D13998	WORD	Память для хранения названий рецептов. Задание 160. Символ 24
D13999	WORD	Память для хранения названий рецептов. Задание 160. Символ 25
D14000	WORD	Память для хранения названий рецептов. Задание 161. Символ 1
D14001	WORD	Память для хранения названий рецептов. Задание 161. Символ 2
D14002	WORD	Память для хранения названий рецептов. Задание 161. Символ 3
D14003	WORD	Память для хранения названий рецептов. Задание 161. Символ 4
D14004	WORD	Память для хранения названий рецептов. Задание 161. Символ 5
D14005	WORD	Память для хранения названий рецептов. Задание 161. Символ 6
D14006	WORD	Память для хранения названий рецептов. Задание 161. Символ 7
D14007	WORD	Память для хранения названий рецептов. Задание 161. Символ 8
D14008	WORD	Память для хранения названий рецептов. Задание 161. Символ 9
D14009	WORD	Память для хранения названий рецептов. Задание 161. Символ 10
D14010	WORD	Память для хранения названий рецептов. Задание 161. Символ 11
D14011	WORD	Память для хранения названий рецептов. Задание 161. Символ 12
D14012	WORD	Память для хранения названий рецептов. Задание 161. Символ 13
D14013	WORD	Память для хранения названий рецептов. Задание 161. Символ 14
D14014	WORD	Память для хранения названий рецептов. Задание 161. Символ 15
D14015	WORD	Память для хранения названий рецептов. Задание 161. Символ 16
D14016	WORD	Память для хранения названий рецептов. Задание 161. Символ 17
D14017	WORD	Память для хранения названий рецептов. Задание 161. Символ 18
D14018	WORD	Память для хранения названий рецептов. Задание 161. Символ 19
D14019	WORD	Память для хранения названий рецептов. Задание 161. Символ 20
D14020	WORD	Память для хранения названий рецептов. Задание 161. Символ 21
D14021	WORD	Память для хранения названий рецептов. Задание 161. Символ 22
D14022	WORD	Память для хранения названий рецептов. Задание 161. Символ 23
D14023	WORD	Память для хранения названий рецептов. Задание 161. Символ 24
D14024	WORD	Память для хранения названий рецептов. Задание 161. Символ 25
D14025	WORD	Память для хранения названий рецептов. Задание 162. Символ 1
D14026	WORD	Память для хранения названий рецептов. Задание 162. Символ 2
D14027	WORD	Память для хранения названий рецептов. Задание 162. Символ 3
D14028	WORD	Память для хранения названий рецептов. Задание 162. Символ 4
D14029	WORD	Память для хранения названий рецептов. Задание 162. Символ 5
D14030	WORD	Память для хранения названий рецептов. Задание 162. Символ 6
D14031	WORD	Память для хранения названий рецептов. Задание 162. Символ 7
D14032	WORD	Память для хранения названий рецептов. Задание 162. Символ 8
D14033	WORD	Память для хранения названий рецептов. Задание 162. Символ 9
D14034	WORD	Память для хранения названий рецептов. Задание 162. Символ 10
D14035	WORD	Память для хранения названий рецептов. Задание 162. Символ 11
D14036	WORD	Память для хранения названий рецептов. Задание 162. Символ 12
D14037	WORD	Память для хранения названий рецептов. Задание 162. Символ 13
D14038	WORD	Память для хранения названий рецептов. Задание 162. Символ 14
D14039	WORD	Память для хранения названий рецептов. Задание 162. Символ 15
D14040	WORD	Память для хранения названий рецептов. Задание 162. Символ 16
D14041	WORD	Память для хранения названий рецептов. Задание 162. Символ 17
D14042	WORD	Память для хранения названий рецептов. Задание 162. Символ 18
D14043	WORD	Память для хранения названий рецептов. Задание 162. Символ 19
D14044	WORD	Память для хранения названий рецептов. Задание 162. Символ 20
D14045	WORD	Память для хранения названий рецептов. Задание 162. Символ 21
D14046	WORD	Память для хранения названий рецептов. Задание 162. Символ 22
D14047	WORD	Память для хранения названий рецептов. Задание 162. Символ 23
D14048	WORD	Память для хранения названий рецептов. Задание 162. Символ 24
D14049	WORD	Память для хранения названий рецептов. Задание 162. Символ 25
D14050	WORD	Память для хранения названий рецептов. Задание 163. Символ 1
D14051	WORD	Память для хранения названий рецептов. Задание 163. Символ 2
D14052	WORD	Память для хранения названий рецептов. Задание 163. Символ 3
D14053	WORD	Память для хранения названий рецептов. Задание 163. Символ 4
D14054	WORD	Память для хранения названий рецептов. Задание 163. Символ 5
D14055	WORD	Память для хранения названий рецептов. Задание 163. Символ 6
D14056	WORD	Память для хранения названий рецептов. Задание 163. Символ 7
D14057	WORD	Память для хранения названий рецептов. Задание 163. Символ 8
D14058	WORD	Память для хранения названий рецептов. Задание 163. Символ 9
D14059	WORD	Память для хранения названий рецептов. Задание 163. Символ 10
D14060	WORD	Память для хранения названий рецептов. Задание 163. Символ 11
D14061	WORD	Память для хранения названий рецептов. Задание 163. Символ 12
D14062	WORD	Память для хранения названий рецептов. Задание 163. Символ 13
D14063	WORD	Память для хранения названий рецептов. Задание 163. Символ 14
D14064	WORD	Память для хранения названий рецептов. Задание 163. Символ 15
D14065	WORD	Память для хранения названий рецептов. Задание 163. Символ 16
D14066	WORD	Память для хранения названий рецептов. Задание 163. Символ 17
D14067	WORD	Память для хранения названий рецептов. Задание 163. Символ 18
D14068	WORD	Память для хранения названий рецептов. Задание 163. Символ 19
D14069	WORD	Память для хранения названий рецептов. Задание 163. Символ 20
D14070	WORD	Память для хранения названий рецептов. Задание 163. Символ 21
D14071	WORD	Память для хранения названий рецептов. Задание 163. Символ 22
D14072	WORD	Память для хранения названий рецептов. Задание 163. Символ 23
D14073	WORD	Память для хранения названий рецептов. Задание 163. Символ 24
D14074	WORD	Память для хранения названий рецептов. Задание 163. Символ 25
D14075	WORD	Память для хранения названий рецептов. Задание 164. Символ 1
D14076	WORD	Память для хранения названий рецептов. Задание 164. Символ 2
D14077	WORD	Память для хранения названий рецептов. Задание 164. Символ 3
D14078	WORD	Память для хранения названий рецептов. Задание 164. Символ 4
D14079	WORD	Память для хранения названий рецептов. Задание 164. Символ 5
D14080	WORD	Память для хранения названий рецептов. Задание 164. Символ 6
D14081	WORD	Память для хранения названий рецептов. Задание 164. Символ 7
D14082	WORD	Память для хранения названий рецептов. Задание 164. Символ 8
D14083	WORD	Память для хранения названий рецептов. Задание 164. Символ 9
D14084	WORD	Память для хранения названий рецептов. Задание 164. Символ 10
D14085	WORD	Память для хранения названий рецептов. Задание 164. Символ 11
D14086	WORD	Память для хранения названий рецептов. Задание 164. Символ 12
D14087	WORD	Память для хранения названий рецептов. Задание 164. Символ 13
D14088	WORD	Память для хранения названий рецептов. Задание 164. Символ 14
D14089	WORD	Память для хранения названий рецептов. Задание 164. Символ 15
D14090	WORD	Память для хранения названий рецептов. Задание 164. Символ 16
D14091	WORD	Память для хранения названий рецептов. Задание 164. Символ 17
D14092	WORD	Память для хранения названий рецептов. Задание 164. Символ 18
D14093	WORD	Память для хранения названий рецептов. Задание 164. Символ 19
D14094	WORD	Память для хранения названий рецептов. Задание 164. Символ 20
D14095	WORD	Память для хранения названий рецептов. Задание 164. Символ 21
D14096	WORD	Память для хранения названий рецептов. Задание 164. Символ 22
D14097	WORD	Память для хранения названий рецептов. Задание 164. Символ 23
D14098	WORD	Память для хранения названий рецептов. Задание 164. Символ 24
D14099	WORD	Память для хранения названий рецептов. Задание 164. Символ 25
D14100	WORD	Память для хранения названий рецептов. Задание 165. Символ 1
D14101	WORD	Память для хранения названий рецептов. Задание 165. Символ 2
D14102	WORD	Память для хранения названий рецептов. Задание 165. Символ 3
D14103	WORD	Память для хранения названий рецептов. Задание 165. Символ 4
D14104	WORD	Память для хранения названий рецептов. Задание 165. Символ 5
D14105	WORD	Память для хранения названий рецептов. Задание 165. Символ 6
D14106	WORD	Память для хранения названий рецептов. Задание 165. Символ 7
D14107	WORD	Память для хранения названий рецептов. Задание 165. Символ 8
D14108	WORD	Память для хранения названий рецептов. Задание 165. Символ 9
D14109	WORD	Память для хранения названий рецептов. Задание 165. Символ 10
D14110	WORD	Память для хранения названий рецептов. Задание 165. Символ 11
D14111	WORD	Память для хранения названий рецептов. Задание 165. Символ 12
D14112	WORD	Память для хранения названий рецептов. Задание 165. Символ 13
D14113	WORD	Память для хранения названий рецептов. Задание 165. Символ 14
D14114	WORD	Память для хранения названий рецептов. Задание 165. Символ 15
D14115	WORD	Память для хранения названий рецептов. Задание 165. Символ 16
D14116	WORD	Память для хранения названий рецептов. Задание 165. Символ 17
D14117	WORD	Память для хранения названий рецептов. Задание 165. Символ 18
D14118	WORD	Память для хранения названий рецептов. Задание 165. Символ 19
D14119	WORD	Память для хранения названий рецептов. Задание 165. Символ 20
D14120	WORD	Память для хранения названий рецептов. Задание 165. Символ 21
D14121	WORD	Память для хранения названий рецептов. Задание 165. Символ 22
D14122	WORD	Память для хранения названий рецептов. Задание 165. Символ 23
D14123	WORD	Память для хранения названий рецептов. Задание 165. Символ 24
D14124	WORD	Память для хранения названий рецептов. Задание 165. Символ 25
D14125	WORD	Память для хранения названий рецептов. Задание 166. Символ 1
D14126	WORD	Память для хранения названий рецептов. Задание 166. Символ 2
D14127	WORD	Память для хранения названий рецептов. Задание 166. Символ 3
D14128	WORD	Память для хранения названий рецептов. Задание 166. Символ 4
D14129	WORD	Память для хранения названий рецептов. Задание 166. Символ 5
D14130	WORD	Память для хранения названий рецептов. Задание 166. Символ 6
D14131	WORD	Память для хранения названий рецептов. Задание 166. Символ 7
D14132	WORD	Память для хранения названий рецептов. Задание 166. Символ 8
D14133	WORD	Память для хранения названий рецептов. Задание 166. Символ 9
D14134	WORD	Память для хранения названий рецептов. Задание 166. Символ 10
D14135	WORD	Память для хранения названий рецептов. Задание 166. Символ 11
D14136	WORD	Память для хранения названий рецептов. Задание 166. Символ 12
D14137	WORD	Память для хранения названий рецептов. Задание 166. Символ 13
D14138	WORD	Память для хранения названий рецептов. Задание 166. Символ 14
D14139	WORD	Память для хранения названий рецептов. Задание 166. Символ 15
D14140	WORD	Память для хранения названий рецептов. Задание 166. Символ 16
D14141	WORD	Память для хранения названий рецептов. Задание 166. Символ 17
D14142	WORD	Память для хранения названий рецептов. Задание 166. Символ 18
D14143	WORD	Память для хранения названий рецептов. Задание 166. Символ 19
D14144	WORD	Память для хранения названий рецептов. Задание 166. Символ 20
D14145	WORD	Память для хранения названий рецептов. Задание 166. Символ 21
D14146	WORD	Память для хранения названий рецептов. Задание 166. Символ 22
D14147	WORD	Память для хранения названий рецептов. Задание 166. Символ 23
D14148	WORD	Память для хранения названий рецептов. Задание 166. Символ 24
D14149	WORD	Память для хранения названий рецептов. Задание 166. Символ 25
D14150	WORD	Память для хранения названий рецептов. Задание 167. Символ 1
D14151	WORD	Память для хранения названий рецептов. Задание 167. Символ 2
D14152	WORD	Память для хранения названий рецептов. Задание 167. Символ 3
D14153	WORD	Память для хранения названий рецептов. Задание 167. Символ 4
D14154	WORD	Память для хранения названий рецептов. Задание 167. Символ 5
D14155	WORD	Память для хранения названий рецептов. Задание 167. Символ 6
D14156	WORD	Память для хранения названий рецептов. Задание 167. Символ 7
D14157	WORD	Память для хранения названий рецептов. Задание 167. Символ 8
D14158	WORD	Память для хранения названий рецептов. Задание 167. Символ 9
D14159	WORD	Память для хранения названий рецептов. Задание 167. Символ 10
D14160	WORD	Память для хранения названий рецептов. Задание 167. Символ 11
D14161	WORD	Память для хранения названий рецептов. Задание 167. Символ 12
D14162	WORD	Память для хранения названий рецептов. Задание 167. Символ 13
D14163	WORD	Память для хранения названий рецептов. Задание 167. Символ 14
D14164	WORD	Память для хранения названий рецептов. Задание 167. Символ 15
D14165	WORD	Память для хранения названий рецептов. Задание 167. Символ 16
D14166	WORD	Память для хранения названий рецептов. Задание 167. Символ 17
D14167	WORD	Память для хранения названий рецептов. Задание 167. Символ 18
D14168	WORD	Память для хранения названий рецептов. Задание 167. Символ 19
D14169	WORD	Память для хранения названий рецептов. Задание 167. Символ 20
D14170	WORD	Память для хранения названий рецептов. Задание 167. Символ 21
D14171	WORD	Память для хранения названий рецептов. Задание 167. Символ 22
D14172	WORD	Память для хранения названий рецептов. Задание 167. Символ 23
D14173	WORD	Память для хранения названий рецептов. Задание 167. Символ 24
D14174	WORD	Память для хранения названий рецептов. Задание 167. Символ 25
D14175	WORD	Память для хранения названий рецептов. Задание 168. Символ 1
D14176	WORD	Память для хранения названий рецептов. Задание 168. Символ 2
D14177	WORD	Память для хранения названий рецептов. Задание 168. Символ 3
D14178	WORD	Память для хранения названий рецептов. Задание 168. Символ 4
D14179	WORD	Память для хранения названий рецептов. Задание 168. Символ 5
D14180	WORD	Память для хранения названий рецептов. Задание 168. Символ 6
D14181	WORD	Память для хранения названий рецептов. Задание 168. Символ 7
D14182	WORD	Память для хранения названий рецептов. Задание 168. Символ 8
D14183	WORD	Память для хранения названий рецептов. Задание 168. Символ 9
D14184	WORD	Память для хранения названий рецептов. Задание 168. Символ 10
D14185	WORD	Память для хранения названий рецептов. Задание 168. Символ 11
D14186	WORD	Память для хранения названий рецептов. Задание 168. Символ 12
D14187	WORD	Память для хранения названий рецептов. Задание 168. Символ 13
D14188	WORD	Память для хранения названий рецептов. Задание 168. Символ 14
D14189	WORD	Память для хранения названий рецептов. Задание 168. Символ 15
D14190	WORD	Память для хранения названий рецептов. Задание 168. Символ 16
D14191	WORD	Память для хранения названий рецептов. Задание 168. Символ 17
D14192	WORD	Память для хранения названий рецептов. Задание 168. Символ 18
D14193	WORD	Память для хранения названий рецептов. Задание 168. Символ 19
D14194	WORD	Память для хранения названий рецептов. Задание 168. Символ 20
D14195	WORD	Память для хранения названий рецептов. Задание 168. Символ 21
D14196	WORD	Память для хранения названий рецептов. Задание 168. Символ 22
D14197	WORD	Память для хранения названий рецептов. Задание 168. Символ 23
D14198	WORD	Память для хранения названий рецептов. Задание 168. Символ 24
D14199	WORD	Память для хранения названий рецептов. Задание 168. Символ 25
D14200	WORD	Память для хранения названий рецептов. Задание 169. Символ 1
D14201	WORD	Память для хранения названий рецептов. Задание 169. Символ 2
D14202	WORD	Память для хранения названий рецептов. Задание 169. Символ 3
D14203	WORD	Память для хранения названий рецептов. Задание 169. Символ 4
D14204	WORD	Память для хранения названий рецептов. Задание 169. Символ 5
D14205	WORD	Память для хранения названий рецептов. Задание 169. Символ 6
D14206	WORD	Память для хранения названий рецептов. Задание 169. Символ 7
D14207	WORD	Память для хранения названий рецептов. Задание 169. Символ 8
D14208	WORD	Память для хранения названий рецептов. Задание 169. Символ 9
D14209	WORD	Память для хранения названий рецептов. Задание 169. Символ 10
D14210	WORD	Память для хранения названий рецептов. Задание 169. Символ 11
D14211	WORD	Память для хранения названий рецептов. Задание 169. Символ 12
D14212	WORD	Память для хранения названий рецептов. Задание 169. Символ 13
D14213	WORD	Память для хранения названий рецептов. Задание 169. Символ 14
D14214	WORD	Память для хранения названий рецептов. Задание 169. Символ 15
D14215	WORD	Память для хранения названий рецептов. Задание 169. Символ 16
D14216	WORD	Память для хранения названий рецептов. Задание 169. Символ 17
D14217	WORD	Память для хранения названий рецептов. Задание 169. Символ 18
D14218	WORD	Память для хранения названий рецептов. Задание 169. Символ 19
D14219	WORD	Память для хранения названий рецептов. Задание 169. Символ 20
D14220	WORD	Память для хранения названий рецептов. Задание 169. Символ 21
D14221	WORD	Память для хранения названий рецептов. Задание 169. Символ 22
D14222	WORD	Память для хранения названий рецептов. Задание 169. Символ 23
D14223	WORD	Память для хранения названий рецептов. Задание 169. Символ 24
D14224	WORD	Память для хранения названий рецептов. Задание 169. Символ 25
D14225	WORD	Память для хранения названий рецептов. Задание 170. Символ 1
D14226	WORD	Память для хранения названий рецептов. Задание 170. Символ 2
D14227	WORD	Память для хранения названий рецептов. Задание 170. Символ 3
D14228	WORD	Память для хранения названий рецептов. Задание 170. Символ 4
D14229	WORD	Память для хранения названий рецептов. Задание 170. Символ 5
D14230	WORD	Память для хранения названий рецептов. Задание 170. Символ 6
D14231	WORD	Память для хранения названий рецептов. Задание 170. Символ 7
D14232	WORD	Память для хранения названий рецептов. Задание 170. Символ 8
D14233	WORD	Память для хранения названий рецептов. Задание 170. Символ 9
D14234	WORD	Память для хранения названий рецептов. Задание 170. Символ 10
D14235	WORD	Память для хранения названий рецептов. Задание 170. Символ 11
D14236	WORD	Память для хранения названий рецептов. Задание 170. Символ 12
D14237	WORD	Память для хранения названий рецептов. Задание 170. Символ 13
D14238	WORD	Память для хранения названий рецептов. Задание 170. Символ 14
D14239	WORD	Память для хранения названий рецептов. Задание 170. Символ 15
D14240	WORD	Память для хранения названий рецептов. Задание 170. Символ 16
D14241	WORD	Память для хранения названий рецептов. Задание 170. Символ 17
D14242	WORD	Память для хранения названий рецептов. Задание 170. Символ 18
D14243	WORD	Память для хранения названий рецептов. Задание 170. Символ 19
D14244	WORD	Память для хранения названий рецептов. Задание 170. Символ 20
D14245	WORD	Память для хранения названий рецептов. Задание 170. Символ 21
D14246	WORD	Память для хранения названий рецептов. Задание 170. Символ 22
D14247	WORD	Память для хранения названий рецептов. Задание 170. Символ 23
D14248	WORD	Память для хранения названий рецептов. Задание 170. Символ 24
D14249	WORD	Память для хранения названий рецептов. Задание 170. Символ 25
D14250	WORD	Память для хранения названий рецептов. Задание 171. Символ 1
D14251	WORD	Память для хранения названий рецептов. Задание 171. Символ 2
D14252	WORD	Память для хранения названий рецептов. Задание 171. Символ 3
D14253	WORD	Память для хранения названий рецептов. Задание 171. Символ 4
D14254	WORD	Память для хранения названий рецептов. Задание 171. Символ 5
D14255	WORD	Память для хранения названий рецептов. Задание 171. Символ 6
D14256	WORD	Память для хранения названий рецептов. Задание 171. Символ 7
D14257	WORD	Память для хранения названий рецептов. Задание 171. Символ 8
D14258	WORD	Память для хранения названий рецептов. Задание 171. Символ 9
D14259	WORD	Память для хранения названий рецептов. Задание 171. Символ 10
D14260	WORD	Память для хранения названий рецептов. Задание 171. Символ 11
D14261	WORD	Память для хранения названий рецептов. Задание 171. Символ 12
D14262	WORD	Память для хранения названий рецептов. Задание 171. Символ 13
D14263	WORD	Память для хранения названий рецептов. Задание 171. Символ 14
D14264	WORD	Память для хранения названий рецептов. Задание 171. Символ 15
D14265	WORD	Память для хранения названий рецептов. Задание 171. Символ 16
D14266	WORD	Память для хранения названий рецептов. Задание 171. Символ 17
D14267	WORD	Память для хранения названий рецептов. Задание 171. Символ 18
D14268	WORD	Память для хранения названий рецептов. Задание 171. Символ 19
D14269	WORD	Память для хранения названий рецептов. Задание 171. Символ 20
D14270	WORD	Память для хранения названий рецептов. Задание 171. Символ 21
D14271	WORD	Память для хранения названий рецептов. Задание 171. Символ 22
D14272	WORD	Память для хранения названий рецептов. Задание 171. Символ 23
D14273	WORD	Память для хранения названий рецептов. Задание 171. Символ 24
D14274	WORD	Память для хранения названий рецептов. Задание 171. Символ 25
D14275	WORD	Память для хранения названий рецептов. Задание 172. Символ 1
D14276	WORD	Память для хранения названий рецептов. Задание 172. Символ 2
D14277	WORD	Память для хранения названий рецептов. Задание 172. Символ 3
D14278	WORD	Память для хранения названий рецептов. Задание 172. Символ 4
D14279	WORD	Память для хранения названий рецептов. Задание 172. Символ 5
D14280	WORD	Память для хранения названий рецептов. Задание 172. Символ 6
D14281	WORD	Память для хранения названий рецептов. Задание 172. Символ 7
D14282	WORD	Память для хранения названий рецептов. Задание 172. Символ 8
D14283	WORD	Память для хранения названий рецептов. Задание 172. Символ 9
D14284	WORD	Память для хранения названий рецептов. Задание 172. Символ 10
D14285	WORD	Память для хранения названий рецептов. Задание 172. Символ 11
D14286	WORD	Память для хранения названий рецептов. Задание 172. Символ 12
D14287	WORD	Память для хранения названий рецептов. Задание 172. Символ 13
D14288	WORD	Память для хранения названий рецептов. Задание 172. Символ 14
D14289	WORD	Память для хранения названий рецептов. Задание 172. Символ 15
D14290	WORD	Память для хранения названий рецептов. Задание 172. Символ 16
D14291	WORD	Память для хранения названий рецептов. Задание 172. Символ 17
D14292	WORD	Память для хранения названий рецептов. Задание 172. Символ 18
D14293	WORD	Память для хранения названий рецептов. Задание 172. Символ 19
D14294	WORD	Память для хранения названий рецептов. Задание 172. Символ 20
D14295	WORD	Память для хранения названий рецептов. Задание 172. Символ 21
D14296	WORD	Память для хранения названий рецептов. Задание 172. Символ 22
D14297	WORD	Память для хранения названий рецептов. Задание 172. Символ 23
D14298	WORD	Память для хранения названий рецептов. Задание 172. Символ 24
D14299	WORD	Память для хранения названий рецептов. Задание 172. Символ 25
D14300	WORD	Память для хранения названий рецептов. Задание 173. Символ 1
D14301	WORD	Память для хранения названий рецептов. Задание 173. Символ 2
D14302	WORD	Память для хранения названий рецептов. Задание 173. Символ 3
D14303	WORD	Память для хранения названий рецептов. Задание 173. Символ 4
D14304	WORD	Память для хранения названий рецептов. Задание 173. Символ 5
D14305	WORD	Память для хранения названий рецептов. Задание 173. Символ 6
D14306	WORD	Память для хранения названий рецептов. Задание 173. Символ 7
D14307	WORD	Память для хранения названий рецептов. Задание 173. Символ 8
D14308	WORD	Память для хранения названий рецептов. Задание 173. Символ 9
D14309	WORD	Память для хранения названий рецептов. Задание 173. Символ 10
D14310	WORD	Память для хранения названий рецептов. Задание 173. Символ 11
D14311	WORD	Память для хранения названий рецептов. Задание 173. Символ 12
D14312	WORD	Память для хранения названий рецептов. Задание 173. Символ 13
D14313	WORD	Память для хранения названий рецептов. Задание 173. Символ 14
D14314	WORD	Память для хранения названий рецептов. Задание 173. Символ 15
D14315	WORD	Память для хранения названий рецептов. Задание 173. Символ 16
D14316	WORD	Память для хранения названий рецептов. Задание 173. Символ 17
D14317	WORD	Память для хранения названий рецептов. Задание 173. Символ 18
D14318	WORD	Память для хранения названий рецептов. Задание 173. Символ 19
D14319	WORD	Память для хранения названий рецептов. Задание 173. Символ 20
D14320	WORD	Память для хранения названий рецептов. Задание 173. Символ 21
D14321	WORD	Память для хранения названий рецептов. Задание 173. Символ 22
D14322	WORD	Память для хранения названий рецептов. Задание 173. Символ 23
D14323	WORD	Память для хранения названий рецептов. Задание 173. Символ 24
D14324	WORD	Память для хранения названий рецептов. Задание 173. Символ 25
D14325	WORD	Память для хранения названий рецептов. Задание 174. Символ 1
D14326	WORD	Память для хранения названий рецептов. Задание 174. Символ 2
D14327	WORD	Память для хранения названий рецептов. Задание 174. Символ 3
D14328	WORD	Память для хранения названий рецептов. Задание 174. Символ 4
D14329	WORD	Память для хранения названий рецептов. Задание 174. Символ 5
D14330	WORD	Память для хранения названий рецептов. Задание 174. Символ 6
D14331	WORD	Память для хранения названий рецептов. Задание 174. Символ 7
D14332	WORD	Память для хранения названий рецептов. Задание 174. Символ 8
D14333	WORD	Память для хранения названий рецептов. Задание 174. Символ 9
D14334	WORD	Память для хранения названий рецептов. Задание 174. Символ 10
D14335	WORD	Память для хранения названий рецептов. Задание 174. Символ 11
D14336	WORD	Память для хранения названий рецептов. Задание 174. Символ 12
D14337	WORD	Память для хранения названий рецептов. Задание 174. Символ 13
D14338	WORD	Память для хранения названий рецептов. Задание 174. Символ 14
D14339	WORD	Память для хранения названий рецептов. Задание 174. Символ 15
D14340	WORD	Память для хранения названий рецептов. Задание 174. Символ 16
D14341	WORD	Память для хранения названий рецептов. Задание 174. Символ 17
D14342	WORD	Память для хранения названий рецептов. Задание 174. Символ 18
D14343	WORD	Память для хранения названий рецептов. Задание 174. Символ 19
D14344	WORD	Память для хранения названий рецептов. Задание 174. Символ 20
D14345	WORD	Память для хранения названий рецептов. Задание 174. Символ 21
D14346	WORD	Память для хранения названий рецептов. Задание 174. Символ 22
D14347	WORD	Память для хранения названий рецептов. Задание 174. Символ 23
D14348	WORD	Память для хранения названий рецептов. Задание 174. Символ 24
D14349	WORD	Память для хранения названий рецептов. Задание 174. Символ 25
D14350	WORD	Память для хранения названий рецептов. Задание 175. Символ 1
D14351	WORD	Память для хранения названий рецептов. Задание 175. Символ 2
D14352	WORD	Память для хранения названий рецептов. Задание 175. Символ 3
D14353	WORD	Память для хранения названий рецептов. Задание 175. Символ 4
D14354	WORD	Память для хранения названий рецептов. Задание 175. Символ 5
D14355	WORD	Память для хранения названий рецептов. Задание 175. Символ 6
D14356	WORD	Память для хранения названий рецептов. Задание 175. Символ 7
D14357	WORD	Память для хранения названий рецептов. Задание 175. Символ 8
D14358	WORD	Память для хранения названий рецептов. Задание 175. Символ 9
D14359	WORD	Память для хранения названий рецептов. Задание 175. Символ 10
D14360	WORD	Память для хранения названий рецептов. Задание 175. Символ 11
D14361	WORD	Память для хранения названий рецептов. Задание 175. Символ 12
D14362	WORD	Память для хранения названий рецептов. Задание 175. Символ 13
D14363	WORD	Память для хранения названий рецептов. Задание 175. Символ 14
D14364	WORD	Память для хранения названий рецептов. Задание 175. Символ 15
D14365	WORD	Память для хранения названий рецептов. Задание 175. Символ 16
D14366	WORD	Память для хранения названий рецептов. Задание 175. Символ 17
D14367	WORD	Память для хранения названий рецептов. Задание 175. Символ 18
D14368	WORD	Память для хранения названий рецептов. Задание 175. Символ 19
D14369	WORD	Память для хранения названий рецептов. Задание 175. Символ 20
D14370	WORD	Память для хранения названий рецептов. Задание 175. Символ 21
D14371	WORD	Память для хранения названий рецептов. Задание 175. Символ 22
D14372	WORD	Память для хранения названий рецептов. Задание 175. Символ 23
D14373	WORD	Память для хранения названий рецептов. Задание 175. Символ 24
D14374	WORD	Память для хранения названий рецептов. Задание 175. Символ 25
D14375	WORD	Память для хранения названий рецептов. Задание 176. Символ 1
D14376	WORD	Память для хранения названий рецептов. Задание 176. Символ 2
D14377	WORD	Память для хранения названий рецептов. Задание 176. Символ 3
D14378	WORD	Память для хранения названий рецептов. Задание 176. Символ 4
D14379	WORD	Память для хранения названий рецептов. Задание 176. Символ 5
D14380	WORD	Память для хранения названий рецептов. Задание 176. Символ 6
D14381	WORD	Память для хранения названий рецептов. Задание 176. Символ 7
D14382	WORD	Память для хранения названий рецептов. Задание 176. Символ 8
D14383	WORD	Память для хранения названий рецептов. Задание 176. Символ 9
D14384	WORD	Память для хранения названий рецептов. Задание 176. Символ 10
D14385	WORD	Память для хранения названий рецептов. Задание 176. Символ 11
D14386	WORD	Память для хранения названий рецептов. Задание 176. Символ 12
D14387	WORD	Память для хранения названий рецептов. Задание 176. Символ 13
D14388	WORD	Память для хранения названий рецептов. Задание 176. Символ 14
D14389	WORD	Память для хранения названий рецептов. Задание 176. Символ 15
D14390	WORD	Память для хранения названий рецептов. Задание 176. Символ 16
D14391	WORD	Память для хранения названий рецептов. Задание 176. Символ 17
D14392	WORD	Память для хранения названий рецептов. Задание 176. Символ 18
D14393	WORD	Память для хранения названий рецептов. Задание 176. Символ 19
D14394	WORD	Память для хранения названий рецептов. Задание 176. Символ 20
D14395	WORD	Память для хранения названий рецептов. Задание 176. Символ 21
D14396	WORD	Память для хранения названий рецептов. Задание 176. Символ 22
D14397	WORD	Память для хранения названий рецептов. Задание 176. Символ 23
D14398	WORD	Память для хранения названий рецептов. Задание 176. Символ 24
D14399	WORD	Память для хранения названий рецептов. Задание 176. Символ 25
D14400	WORD	Память для хранения названий рецептов. Задание 177. Символ 1
D14401	WORD	Память для хранения названий рецептов. Задание 177. Символ 2
D14402	WORD	Память для хранения названий рецептов. Задание 177. Символ 3
D14403	WORD	Память для хранения названий рецептов. Задание 177. Символ 4
D14404	WORD	Память для хранения названий рецептов. Задание 177. Символ 5
D14405	WORD	Память для хранения названий рецептов. Задание 177. Символ 6
D14406	WORD	Память для хранения названий рецептов. Задание 177. Символ 7
D14407	WORD	Память для хранения названий рецептов. Задание 177. Символ 8
D14408	WORD	Память для хранения названий рецептов. Задание 177. Символ 9
D14409	WORD	Память для хранения названий рецептов. Задание 177. Символ 10
D14410	WORD	Память для хранения названий рецептов. Задание 177. Символ 11
D14411	WORD	Память для хранения названий рецептов. Задание 177. Символ 12
D14412	WORD	Память для хранения названий рецептов. Задание 177. Символ 13
D14413	WORD	Память для хранения названий рецептов. Задание 177. Символ 14
D14414	WORD	Память для хранения названий рецептов. Задание 177. Символ 15
D14415	WORD	Память для хранения названий рецептов. Задание 177. Символ 16
D14416	WORD	Память для хранения названий рецептов. Задание 177. Символ 17
D14417	WORD	Память для хранения названий рецептов. Задание 177. Символ 18
D14418	WORD	Память для хранения названий рецептов. Задание 177. Символ 19
D14419	WORD	Память для хранения названий рецептов. Задание 177. Символ 20
D14420	WORD	Память для хранения названий рецептов. Задание 177. Символ 21
D14421	WORD	Память для хранения названий рецептов. Задание 177. Символ 22
D14422	WORD	Память для хранения названий рецептов. Задание 177. Символ 23
D14423	WORD	Память для хранения названий рецептов. Задание 177. Символ 24
D14424	WORD	Память для хранения названий рецептов. Задание 177. Символ 25
D14425	WORD	Память для хранения названий рецептов. Задание 178. Символ 1
D14426	WORD	Память для хранения названий рецептов. Задание 178. Символ 2
D14427	WORD	Память для хранения названий рецептов. Задание 178. Символ 3
D14428	WORD	Память для хранения названий рецептов. Задание 178. Символ 4
D14429	WORD	Память для хранения названий рецептов. Задание 178. Символ 5
D14430	WORD	Память для хранения названий рецептов. Задание 178. Символ 6
D14431	WORD	Память для хранения названий рецептов. Задание 178. Символ 7
D14432	WORD	Память для хранения названий рецептов. Задание 178. Символ 8
D14433	WORD	Память для хранения названий рецептов. Задание 178. Символ 9
D14434	WORD	Память для хранения названий рецептов. Задание 178. Символ 10
D14435	WORD	Память для хранения названий рецептов. Задание 178. Символ 11
D14436	WORD	Память для хранения названий рецептов. Задание 178. Символ 12
D14437	WORD	Память для хранения названий рецептов. Задание 178. Символ 13
D14438	WORD	Память для хранения названий рецептов. Задание 178. Символ 14
D14439	WORD	Память для хранения названий рецептов. Задание 178. Символ 15
D14440	WORD	Память для хранения названий рецептов. Задание 178. Символ 16
D14441	WORD	Память для хранения названий рецептов. Задание 178. Символ 17
D14442	WORD	Память для хранения названий рецептов. Задание 178. Символ 18
D14443	WORD	Память для хранения названий рецептов. Задание 178. Символ 19
D14444	WORD	Память для хранения названий рецептов. Задание 178. Символ 20
D14445	WORD	Память для хранения названий рецептов. Задание 178. Символ 21
D14446	WORD	Память для хранения названий рецептов. Задание 178. Символ 22
D14447	WORD	Память для хранения названий рецептов. Задание 178. Символ 23
D14448	WORD	Память для хранения названий рецептов. Задание 178. Символ 24
D14449	WORD	Память для хранения названий рецептов. Задание 178. Символ 25
D14450	WORD	Память для хранения названий рецептов. Задание 179. Символ 1
D14451	WORD	Память для хранения названий рецептов. Задание 179. Символ 2
D14452	WORD	Память для хранения названий рецептов. Задание 179. Символ 3
D14453	WORD	Память для хранения названий рецептов. Задание 179. Символ 4
D14454	WORD	Память для хранения названий рецептов. Задание 179. Символ 5
D14455	WORD	Память для хранения названий рецептов. Задание 179. Символ 6
D14456	WORD	Память для хранения названий рецептов. Задание 179. Символ 7
D14457	WORD	Память для хранения названий рецептов. Задание 179. Символ 8
D14458	WORD	Память для хранения названий рецептов. Задание 179. Символ 9
D14459	WORD	Память для хранения названий рецептов. Задание 179. Символ 10
D14460	WORD	Память для хранения названий рецептов. Задание 179. Символ 11
D14461	WORD	Память для хранения названий рецептов. Задание 179. Символ 12
D14462	WORD	Память для хранения названий рецептов. Задание 179. Символ 13
D14463	WORD	Память для хранения названий рецептов. Задание 179. Символ 14
D14464	WORD	Память для хранения названий рецептов. Задание 179. Символ 15
D14465	WORD	Память для хранения названий рецептов. Задание 179. Символ 16
D14466	WORD	Память для хранения названий рецептов. Задание 179. Символ 17
D14467	WORD	Память для хранения названий рецептов. Задание 179. Символ 18
D14468	WORD	Память для хранения названий рецептов. Задание 179. Символ 19
D14469	WORD	Память для хранения названий рецептов. Задание 179. Символ 20
D14470	WORD	Память для хранения названий рецептов. Задание 179. Символ 21
D14471	WORD	Память для хранения названий рецептов. Задание 179. Символ 22
D14472	WORD	Память для хранения названий рецептов. Задание 179. Символ 23
D14473	WORD	Память для хранения названий рецептов. Задание 179. Символ 24
D14474	WORD	Память для хранения названий рецептов. Задание 179. Символ 25
D14475	WORD	Память для хранения названий рецептов. Задание 180. Символ 1
D14476	WORD	Память для хранения названий рецептов. Задание 180. Символ 2
D14477	WORD	Память для хранения названий рецептов. Задание 180. Символ 3
D14478	WORD	Память для хранения названий рецептов. Задание 180. Символ 4
D14479	WORD	Память для хранения названий рецептов. Задание 180. Символ 5
D14480	WORD	Память для хранения названий рецептов. Задание 180. Символ 6
D14481	WORD	Память для хранения названий рецептов. Задание 180. Символ 7
D14482	WORD	Память для хранения названий рецептов. Задание 180. Символ 8
D14483	WORD	Память для хранения названий рецептов. Задание 180. Символ 9
D14484	WORD	Память для хранения названий рецептов. Задание 180. Символ 10
D14485	WORD	Память для хранения названий рецептов. Задание 180. Символ 11
D14486	WORD	Память для хранения названий рецептов. Задание 180. Символ 12
D14487	WORD	Память для хранения названий рецептов. Задание 180. Символ 13
D14488	WORD	Память для хранения названий рецептов. Задание 180. Символ 14
D14489	WORD	Память для хранения названий рецептов. Задание 180. Символ 15
D14490	WORD	Память для хранения названий рецептов. Задание 180. Символ 16
D14491	WORD	Память для хранения названий рецептов. Задание 180. Символ 17
D14492	WORD	Память для хранения названий рецептов. Задание 180. Символ 18
D14493	WORD	Память для хранения названий рецептов. Задание 180. Символ 19
D14494	WORD	Память для хранения названий рецептов. Задание 180. Символ 20
D14495	WORD	Память для хранения названий рецептов. Задание 180. Символ 21
D14496	WORD	Память для хранения названий рецептов. Задание 180. Символ 22
D14497	WORD	Память для хранения названий рецептов. Задание 180. Символ 23
D14498	WORD	Память для хранения названий рецептов. Задание 180. Символ 24
D14499	WORD	Память для хранения названий рецептов. Задание 180. Символ 25
D00129	WORD	Фиксированное число 129
D00132	WORD	Фиксированное число 132
D00133	WORD	Фиксированное число 133
D00134	WORD	Фиксированное число 134
D00135	WORD	Фиксированное число 135
D00136	WORD	Фиксированное число 136
D00137	WORD	Фиксированное число 137
D00138	WORD	Фиксированное число 138
D00139	WORD	Фиксированное число 139
D00140	WORD	Фиксированное число 140
D00141	WORD	Фиксированное число 141
D00142	WORD	Фиксированное число 142
D00143	WORD	Фиксированное число 143
D00144	WORD	Фиксированное число 144
D00145	WORD	Фиксированное число 145
D00146	WORD	Фиксированное число 146
D00147	WORD	Фиксированное число 147
D00148	WORD	Фиксированное число 148
D00149	WORD	Фиксированное число 149
D00150	WORD	Фиксированное число 150
D00151	WORD	Фиксированное число 151
D00152	WORD	Фиксированное число 152
D00153	WORD	Фиксированное число 153
D00154	WORD	Фиксированное число 154
D00155	WORD	Фиксированное число 155
D00156	WORD	Фиксированное число 156
D00157	WORD	Фиксированное число 157
D00158	WORD	Фиксированное число 158
D00159	WORD	Фиксированное число 159
D00160	WORD	Фиксированное число 160
D00161	WORD	Фиксированное число 161
D00162	WORD	Фиксированное число 162
D00163	WORD	Фиксированное число 163
D00164	WORD	Фиксированное число 164
D00165	WORD	Фиксированное число 165
D00166	WORD	Фиксированное число 166
D00167	WORD	Фиксированное число 167
D00168	WORD	Фиксированное число 168
D00169	WORD	Фиксированное число 169
D00170	WORD	Фиксированное число 170
D00171	WORD	Фиксированное число 171
D00172	WORD	Фиксированное число 172
D00173	WORD	Фиксированное число 173
D00174	WORD	Фиксированное число 174
D00175	WORD	Фиксированное число 175
D00176	WORD	Фиксированное число 176
D00177	WORD	Фиксированное число 177
D00178	WORD	Фиксированное число 178
D00179	WORD	Фиксированное число 179
D00180	WORD	Фиксированное число 180
D00181	WORD	Фиксированное число 181
D00182	WORD	Фиксированное число 182
D00183	WORD	Фиксированное число 183
D00184	WORD	Фиксированное число 184
D00185	WORD	Фиксированное число 185
D00186	WORD	Фиксированное число 186
D00187	WORD	Фиксированное число 187
D00188	WORD	Фиксированное число 188
D00189	WORD	Фиксированное число 189
D00190	WORD	Фиксированное число 190
D00191	WORD	Фиксированное число 191
D00192	WORD	Фиксированное число 192
D00193	WORD	Фиксированное число 193
D00194	WORD	Фиксированное число 194
D00195	WORD	Фиксированное число 195
D00196	WORD	Фиксированное число 196
D00197	WORD	Фиксированное число 197
D00198	WORD	Фиксированное число 198
D00200	WORD	Фиксированное число 200
D00252	WORD	MULNULL
D00253	WORD	MULNULL
D00254	WORD	MULNULL
D00257	WORD	MULNULL
D00258	WORD	MULNULL
D00259	WORD	MULNULL
D00261	WORD	MULNULL
D00262	WORD	MULNULL
D00263	WORD	MULNULL
D19001	WORD	Редактируемое имя задания. Символ 2
D19002	WORD	Редактируемое имя задания. Символ 3
D19003	WORD	Редактируемое имя задания. Символ 4
D19004	WORD	Редактируемое имя задания. Символ 5
D19005	WORD	Редактируемое имя задания. Символ 6
D19006	WORD	Редактируемое имя задания. Символ 7
D19007	WORD	Редактируемое имя задания. Символ 8
D19008	WORD	Редактируемое имя задания. Символ 9
D19009	WORD	Редактируемое имя задания. Символ 10
D19010	WORD	Редактируемое имя задания. Символ 11
D19011	WORD	Редактируемое имя задания. Символ 12
D19012	WORD	Редактируемое имя задания. Символ 13
D19013	WORD	Редактируемое имя задания. Символ 14
D19014	WORD	Редактируемое имя задания. Символ 15
D19015	WORD	Редактируемое имя задания. Символ 16
D19016	WORD	Редактируемое имя задания. Символ 17
D19017	WORD	Редактируемое имя задания. Символ 18
D19018	WORD	Редактируемое имя задания. Символ 19
D19019	WORD	Редактируемое имя задания. Символ 20
D19020	WORD	Редактируемое имя задания. Символ 21
D19021	WORD	Редактируемое имя задания. Символ 22
D19022	WORD	Редактируемое имя задания. Символ 23
D19023	WORD	Редактируемое имя задания. Символ 24
D19024	WORD	Редактируемое имя задания. Символ 25
D00510	WORD	Количество рядов на пластине
D00511	WORD	Количество ячеек в нечётных рядах
D00512	WORD	Количество ячеек в чётных рядах
D00517	WORD	Кондуктор, шаг для установки ячеек в ряду
D00518	WORD	Кондуктор, шаг для установки между рядами
P11150	BIT	Двойной захват, захват 1, L1 (0)
P11160	BIT	Двойной захват, захват 1, l1
P11170	BIT	Двойной захват, захват 2, L2
P11180	BIT	Двойной захват, захват 2, l2
P11190	BIT	Параллельнй захват, длина L
P11200	BIT	Параллельнй захват, длина l
P11210	BIT	Патрон, длина L
P11220	BIT	Патрон, длина l
P11240	BIT	Расстояние между ячейками
P11250	BIT	Расстояние между рядами
P11260	BIT	Смещение чётного ряда
P11280	BIT	Заготовка. Втулка. L1
P11290	BIT	Заготовка. Втулка. L2
P11300	BIT	Заготовка. Вал L11
P11310	BIT	Заготовка. Вал L12
P11320	BIT	Заготовка. Вал L13
P11330	BIT	Заготовка. Вал H1
P11340	BIT	Заготовка. Вал D1
P11350	BIT	Заготовка. Вал L21
P11360	BIT	Заготовка. Вал L22
P11370	BIT	Заготовка. Вал L23
P11380	BIT	Заготовка. Вал H2
P11390	BIT	Заготовка. Вал D2
P11400	BIT	Номер станции перехвата при развороте втулуи
P11410	BIT	Поправка по высоте при развороте втулки
P11420	BIT	Заготовка. Втулка. D1
P11430	BIT	Заготовка. Втулка. D2
P11440	BIT	Кондуктор, расстояние от центра ячейки до стенки
P1000D	BIT	Робот в режиме отладки
P10060	BIT	Состояние двойного захвата 1
P10070	BIT	Состояние двойного захвата 2
P10080	BIT	Состояние параллельного захвата
P10090	BIT	Состояние патрона
P10100	BIT	Состояние станции перехвата
P10110	BIT	Обработано деталей
P10120	BIT	Следующая деталь
P10130	BIT	Код ошибки на роботе
P1100	WORD	Включить моторы на роботе
P1101	WORD	Открыть захват 1
P1102	WORD	Патрон 1 открыт
P1103	WORD	Запустить задание на роботе
P1104	WORD	Полка 1 включена
P1106	WORD	Скорость робота
P1107	WORD	Прижим при захвате детали с полки
P1108	WORD	Прижим при захвате детали из патрона
P1109	WORD	Прижим при установке детали в призмы
P1110	WORD	Время открытия двойного захвата 1
P1111	WORD	Время открытия двойного захвата 2
P1112	WORD	Время открытия параллельного захвата
P1113	WORD	Номер задания
P1114	WORD	Разворот детали перед установкой в патрон
P1123	WORD	Количество рядов на пластине
P1127	WORD	Кондуктор, шаг для установки ячеек в ряду
P1000	WORD	Моторы робота включены
P1001	WORD	Захват 1 открыт
P1002	WORD	Открыть патрон 1
P1003	WORD	Робот готов к запуску задания
P1004	WORD	Полка 1 открыта
P1005	WORD	Переключение зоны безопасности на лидаре
P1014	WORD	Двойной захват. Захват 1 пустой
P1015	WORD	Станция перехвата. Пустая
D00537.0	BIT	Номер станции перехвата при развороте втулуи
D00538.0	BIT	Поправка по высоте при развороте втулки
M00209	BIT	Требуется запуск задания
T0021	BIT/WORD	T100MS Время сброса задания
D00340	WORD	Прижим для полки
D00341	WORD	Прижим для станка
D00342	WORD	Прижим для перехвата
M0011B	BIT	HMI: Возврат робота в домашнее положение
P11032	BIT	Робота в домашнее положение
D00240	WORD	Пароль HMI
D00241	WORD	Пароль HMI
D00314	WORD	Отображение количества деталей